INTERFACE I_MessageData

PROPERTY DirRoot : POINTER to string(255)
SET
END_SET
END_PROPERTY

PROPERTY ErrorIndex : reference to uint
SET
END_SET
END_PROPERTY

PROPERTY FileRoot : pointer to string(255)
SET
END_SET
END_PROPERTY

PROPERTY LocalTime : pointer to DT
SET
END_SET
END_PROPERTY

PROPERTY MessageIndex : reference to uint
SET
END_SET
END_PROPERTY

PROPERTY MsgList : pointer to ARRAY[1..GVL_MSG.MAX_MESSAGE] OF st_message
SET
END_SET
END_PROPERTY

END_INTERFACE

(* stored: Version 1.1.0.1, ProductVersion 3.1.4026.13
   Itf I_MessageData: Id {678edade-56f5-42ee-b605-315d17aa32d8}
   Property DirRoot: Id {72e09ed6-4fdd-4696-92d8-080ae20ec4d9}
   Set Set: Id {0dd7faec-9c04-4d12-965c-f25f8b9b01ed}
   Property ErrorIndex: Id {4b4f855a-4bb4-4656-906a-bf1374fa42a5}
   Set Set: Id {8987722d-a6c5-4f0c-b1b7-226d789b1b69}
   Property FileRoot: Id {66eced91-0c49-4bf2-ad71-cb1623cd4592}
   Set Set: Id {ef65b947-8cad-4457-901d-feb68e2197f0}
   Property LocalTime: Id {f329ddc8-ea03-4a4a-ae7e-9bd7834120bf}
   Set Set: Id {7e23dafa-56c5-4bd0-aeff-573a168f9dd9}
   Property MessageIndex: Id {bad99a9f-5aa2-4377-b0d5-cc1d69964861}
   Set Set: Id {478bf889-0881-4475-b6d9-80d3a1eae5ea}
   Property MsgList: Id {c1d0d785-60d1-4b22-a561-8d64b4b2aaa7}
   Set Set: Id {8e730aa0-4f63-4a54-9cd5-abe31da80a7c} *)
